(*********************************** G.D S.p.A. - Technical Department ***********************************
============= PROGRAM INFO ============
FOLDER:             TBD
MACHINES INVOLVED:  TBD 

============= DESCRIPTION =============
csp machine declaration

============= REVISIONS ===============
Date		Version	 	Author      	Description             
----------	-------		------------  	--------------------------------------------
2019/04/05 	0000.00	 	M.Grasso		Creation of the PRG

**********************************************************************************************************)
(*$R process_ref := prc; $*)
PROGRAM csp_case_feed_magazine_ls_belt
VAR
		
	prc:											process;
	prc_path:										STRING;
	
	axis:											axis;
	
	actual_velocity_mms:							LREAL:=0.0;
	velocity_req_mms:								LREAL:=0.0;
	ready:											BOOL:=FALSE;

	disabled:										BOOL:=FALSE;
		
	velocity_req_limited_mms:						LREAL:= 0.0;
	override_percent:								REAL:= 0.0; (*$P $*)

	fsm_enable_condition:							BOOL;
	fsm_status:										csp_caser_feed_magazine_ls_belt_status_enum;
	fsm_log:										fsm;
	torque_limit:									INT := 2000;    (*$P $*)
	torque_limit_old:								INT;	
	belt_speed: 									LREAL := 10;
	servo_on_condition: 							BOOL;
	enable_delay: TON;
	Torque_force_constant: 							LREAL := 0.47;
END_VAR

VAR_INPUT

	i_downstream_ready:								BOOL;(*$M desc := Downstream Process Ready; $*)
	i_upstream_running:								BOOL;
	i_upstream_velocity:							LREAL;
	disable_req:									BOOL:=FALSE;
	fault_bool:										BOOL:=FALSE;
END_VAR

VAR CONSTANT
	
	CONSTANTS:										csp_case_feed_magazine_constant_struct;
	
END_VAR

_read_var_input();

_object_manager();

IF NOT objects_running()
THEN
	RETURN;	
END_IF

_read_process_image();

_mode_manager();

CASE process_get_mode(prc) OF
	MODE_ABSENT:
		IF axis_get_mode(axis) = MODE_TEST
		THEN
			safety_integrated_series_close(csp_case_main_safety_drives_SD8400.chB_smes_sis);
		END_IF
		RETURN;
	MODE_INACTIVE:
		RETURN;
	MODE_TEST:
		_handle_process_test();
END_CASE

_set_runtime_properties();

(********************************* BODY *********************************)
(************************************************************************)
axis.actual_torque := (axis.actual_current * Torque_force_constant)/1000;

fsm_enable_condition :=	NOT disable_req
						AND
						NOT fault_bool
						AND
						axis_is_ok(FALSE, axis)
						AND
						process_is_ready(prc)
						AND
						process_subtree_is_ready(prc)
						AND NOT 
						csp_main_accuchange.Brand_Change_Occurred
						AND
						servo_on_condition;


IF	NOT fsm_enable_condition
	AND
	fsm_status <> CSP_CASE_FEED_MAGAZINE_LS_BELT_STATUS_DISABLED
	AND
	fsm_status < CSP_CASE_FEED_MAGAZINE_LS_BELT_STATUS_STOP_REQUEST
THEN
	fsm_status	:=	CSP_CASE_FEED_MAGAZINE_LS_BELT_STATUS_DISABLE_REQUEST;
END_IF

velocity_req_mms := i_upstream_velocity * (100 + override_percent) / 100;

IF torque_limit <> Torque_limit_old
THEN
	 IF soe_drive_channel_write_parameter(
		channel:=csp_case_feed_magazine_ls_belt.axis.soe_drive_channel, 
		idn:= S_0_IDN + 92, 
		data_element:=soe_drive_element_value , 
		data_source:= ADR(torque_limit), 
		data_lenght:= SIZEOF(torque_limit), 
		CONVERSION_this:= csp_case_feed_magazine_ls_belt.axis.soe_drive^)= SOE_DRIVE_RETURN_VALUE_DONE
	THEN 
		torque_limit_old := Torque_limit;
	END_IF
END_IF
	
CASE fsm_status OF
	
	CSP_CASE_FEED_MAGAZINE_LS_BELT_STATUS_NOT_INITIALIZED:
	
        IF	axis_is_ok(return_when_absent := TRUE, CONVERSION_this := axis)
        THEN
            fsm_status := CSP_CASE_FEED_MAGAZINE_LS_BELT_STATUS_DISABLED;
        END_IF

		
	CSP_CASE_FEED_MAGAZINE_LS_BELT_STATUS_DISABLED:
	
		IF	fsm_enable_condition
		THEN
			fsm_status := CSP_CASE_FEED_MAGAZINE_LS_BELT_STATUS_ENABLE_REQUEST;
		END_IF;

		
	CSP_CASE_FEED_MAGAZINE_LS_BELT_STATUS_ENABLE_REQUEST:
	
 	   	axis_enable(axis);
		IF axis_enable(axis)
		THEN
			axis_set_override(
				speed_override_percent 	:= 0,
				CONVERSION_this 					:= axis);
				
			fsm_status	:=	CSP_CASE_FEED_MAGAZINE_LS_BELT_STATUS_ENABLING;
		END_IF;
		

	CSP_CASE_FEED_MAGAZINE_LS_BELT_STATUS_ENABLING:
	
		IF	axis_is_standstill(axis)
			THEN
			fsm_status	:=	CSP_CASE_FEED_MAGAZINE_LS_BELT_STATUS_ENABLED;
		END_IF;

		
	CSP_CASE_FEED_MAGAZINE_LS_BELT_STATUS_ENABLED:

		velocity_req_limited_mms := velocity_req_mms;
		velocity_req_limited_mms := MAX(velocity_req_limited_mms, CONSTANTS.MIN_VELOCITY_MMpSEC);
		velocity_req_limited_mms := MIN(velocity_req_limited_mms, CONSTANTS.MAX_VELOCITY_MMpSEC);

		IF filter_is_off(csp_case_feed_magazine_ls_sensors.feed_di_flt)
			THEN				
				IF axis_move_velocity(
					velocity		:=	belt_speed,//MOTOR_MAX_VELOCITY_DEGPS,
					acceleration	:= CONSTANTS.RUNNING_ACCELERATION_MMMpSEC2, 
					deceleration	:= CONSTANTS.RUNNING_DECELERATION_MMpSEC2, 
					jerk			:= CONSTANTS.RUNNING_JERK_MMpSEC3,
					buffer_mode		:=	AXIS_BUFFER_MODE_ABORTING,
					CONVERSION_this			:=	axis)
					
				THEN
					fsm_status	:=	CSP_CASE_FEED_MAGAZINE_LS_BELT_STATUS_RUNNING;
				END_IF
		END_IF


	CSP_CASE_FEED_MAGAZINE_LS_BELT_STATUS_RUNNING:
	
		IF 	(filter_is_on(csp_case_feed_magazine_ls_sensors.feed_di_flt) //prox met and on for X amount of ms entered in filter
			OR		
				(
					csp_case_feed_kinematic.x_actual_position < -940 //Position in X when case EOAT at PICK positon
					AND NOT motorization_conditioner_is_active(csp_case_feed_magazine.magazine_not_primed_motcond)
				)
			)
			OR message_is_on(csp_case_feed_magazine.ls_magazine_run_limit_aem)
		THEN
			axis_set_override(
				speed_override_percent 	:= 0,
				CONVERSION_this 		:= axis);
		ELSE
			axis_set_override(
				speed_override_percent 	:= 100,
				CONVERSION_this 		:= axis);
		END_IF
	
		
	CSP_CASE_FEED_MAGAZINE_LS_BELT_STATUS_STOP_REQUEST:

		axis_stop(
		    deceleration 		:= CONSTANTS.RUNNING_DECELERATION_MMpSEC2,
		    jerk 				:= CONSTANTS.MAX_JERK_MMpSEC3,
		    CONVERSION_this 	:= axis);

		IF 	axis_is_standstill(axis)
			OR
			NOT axis_is_ok(FALSE, axis)
			OR
			axis_is_disabled(axis)
		THEN
			fsm_status := CSP_CASE_FEED_MAGAZINE_LS_BELT_STATUS_DISABLE_REQUEST;
		END_IF

		
	CSP_CASE_FEED_MAGAZINE_LS_BELT_STATUS_DISABLE_REQUEST:
	
   		axis_disable(axis);
   		fsm_status := CSP_CASE_FEED_MAGAZINE_LS_BELT_STATUS_DISABLING;

		
	CSP_CASE_FEED_MAGAZINE_LS_BELT_STATUS_DISABLING:
	
        IF	axis_is_disabled(axis)
        THEN
            fsm_status := CSP_CASE_FEED_MAGAZINE_LS_BELT_STATUS_DISABLED;
        END_IF;

END_CASE;

(************************************************************************)
(************************************************************************)

_handle_messages();

_write_output();

ACTION _handle_messages:
;
END_ACTION

ACTION _handle_process_test:
;
END_ACTION

ACTION _mode_manager:
IF process_mode_req_is_pending(prc)
THEN
    process_apply_mode_req_first_step(prc);
    CASE process_get_mode(prc) OF
        MODE_TO_ABSENT:
			;
        MODE_TO_INACTIVE:
			;
        MODE_TO_TEST:
			;
        MODE_TO_OPERATIONAL:
			;
    END_CASE
    process_apply_mode_req_second_step(prc);
END_IF
END_ACTION

ACTION _object_manager:
IF objects_initialization()
THEN
	sub_process_init(	
		object_name									:= 'csp_case_feed_magazine_ls_belt.prc', 
		process										:= csp_case_feed_magazine_ls.prc, 
		CONVERSION_this								:= prc);
		
	prc_path 										:= process_get_path(prc);
	
(* axis smes *)
	IF csp_main_configurator.Physical_hw
	THEN
	
		axis_init(
			object_name								:= CONCAT(prc_path, '_axis'), 
			axis_type								:= AXIS_TYPE_SERVO, 
			encoder_scaling_factor					:= G_SERVO_ENCODER_SCALING_FACTOR_DEGPINC,
			modulo									:= G_MODULO_360_DEG, 
			process									:= prc, 
			CONVERSION_this							:= axis);
			
		axis_add_safety_integrated_series(
			safety_integrated_series 				:= csp_case_main_safety_drives_SD8400.chB_smes_sis,
			CONVERSION_this							:= axis);
		
	ELSE
		axis_init(
			object_name								:= CONCAT(prc_path, '_axis'), 
			axis_type								:= AXIS_TYPE_VIRTUAL, 
			encoder_scaling_factor					:= G_VIRTUAL_ENCODER_SCALING_FACTOR_DEGPINC,
			modulo									:= G_MODULO_360_DEG, 
			process									:= prc, 
			CONVERSION_this							:= axis);		
				
	END_IF
	
	axis_set_max_dynamic(
		reference_velocity							:=	CONSTANTS.MOTOR_MAX_VELOCITY_DEGPS,
		velocity									:=	CONSTANTS.MOTOR_MAX_VELOCITY_DEGPS,
		acceleration								:=	CONSTANTS.MOTOR_MAX_ACCELERATION_DEGPS2,
		deceleration								:=	CONSTANTS.MOTOR_MAX_DECELERATION_DEGPS2,
		jerk										:=	CONSTANTS.MOTOR_MAX_JERK_DEGPS3,
		following_error								:=	CONSTANTS.MOTOR_MAX_FOLLOWING_ERROR_DEG,
		CONVERSION_this								:=	axis);
		
	axis_add_soe_drive(
		channel										:=	SOE_DRIVE_CHANNEL_B,
		soe_drive									:=	csp_case_main_drives.SD8400_drv,
		CONVERSION_this								:=	axis);


END_IF

IF objects_running()
THEN
	process_cycle(prc);
	axis_cycle(axis);
END_IF
END_ACTION

ACTION _read_process_image:
;
END_ACTION

ACTION _read_var_input:
;
END_ACTION

ACTION _set_runtime_properties:
enable_delay(IN:=axis_is_ready_to_enable(axis) , PT:=T#2S , Q=> servo_on_condition , ET=> );
END_ACTION

ACTION _write_output:
;
END_ACTION

END_PROGRAM

(* stored: Version 1.1.0.1, ProductVersion 3.1.4024.3
   POU csp_case_feed_magazine_ls_belt: Id {cfe9a2e6-1b53-4156-9c00-1de635c46d1f}, SpecialFunc None
   Action _handle_messages: Id {e8f6bd8e-25d9-4e1c-b9fc-0e14d8900411}
   Action _handle_process_test: Id {f823141e-f610-4b4c-892f-9beb9b0d0329}
   Action _mode_manager: Id {30aa2f13-c2f0-42e6-a0fd-048c3f0eb0f2}
   Action _object_manager: Id {4b6d992a-d10a-4ed5-b46d-a7e2842fd24a}
   Action _read_process_image: Id {519aafff-e6d5-4e1d-a639-64e4fa5aa2de}
   Action _read_var_input: Id {762f50ec-366a-48f7-a79f-193a727ed435}
   Action _set_runtime_properties: Id {db52eb60-33d9-4724-812c-304c321568fd}
   Action _write_output: Id {d157c75c-77fa-40f5-b4be-8220a1440191} *)
